FUNCTION getInBolDebounced : BOOL
VAR_INPUT
	bol_GlobalEnableForce: BOOL;
	udiSample_ms: UDINT;		// Sample time from me.FUBInfo.udiSample_ms
	udiDebounceTime_ms: UDINT;	// Wait time for debouncing in ms
	p_Input: POINTER TO T_Ctrl_IoBoolDebounced;
END_VAR

// The input is accepted only after the debounce time (udiDebounceTime_ms)
// If the signal changes during this time, the timer will be restarted

p_Input^.state := p_Input^.map;

IF (p_Input^.EnForce AND bol_GlobalEnableForce) THEN	// Forced signal, no debouncing neccessary
	p_Input^.intern := p_Input^.force;
ELSE													// Debounce signal
	IF p_Input^.intern <> p_Input^.map THEN
		p_Input^.udinDebouncedTimeCounter_ms := 0;
	END_IF
	IF p_Input^.udinDebouncedTimeCounter_ms < udiDebounceTime_ms THEN
		p_Input^.udinDebouncedTimeCounter_ms := p_Input^.udinDebouncedTimeCounter_ms + udiSample_ms;
	ELSE
		p_Input^.intern := p_Input^.map;		
	END_IF
END_IF;

getInBolDebounced := p_Input^.intern;

END_FUNCTION

(* stored: Version 1.1.0.1, ProductVersion 3.1.0.19
   POU getInBolDebounced: Id {bfc9701f-c020-475a-8a42-2ecab51c9483} *)
